INTERFACE I_DeserializerObjectForwardEnumerator EXTENDS I_Disposable

PROPERTY PUBLIC Current : I_Deserializer
GET
END_GET
END_PROPERTY

PROPERTY IsValid : BOOL
GET
END_GET
END_PROPERTY

PROPERTY Key : T_MAXSTRING
GET
END_GET
END_PROPERTY

METHOD MoveNext : BOOL
VAR_INPUT
END_VAR
END_METHOD

END_INTERFACE

(* stored: Version 1.1.0.1, ProductVersion 3.1.4024.12
   Itf I_DeserializerObjectForwardEnumerator: Id {4aa77d71-92a4-036e-397e-318ade50e4f8}
   Property Current: Id {c85a0a2e-7ad5-0667-211d-0f0eb5551b1d}
   Get Get: Id {dc71cbed-b22a-06bb-1cde-d3cef839c8cc}
   Property IsValid: Id {e0b342ed-ea59-00ab-0145-3d582b50d050}
   Get Get: Id {1adcd0c0-e8e5-03ae-0d04-9d5bad6bb5fd}
   Property Key: Id {166b0429-2001-0abb-3b8a-e0bee278bcc5}
   Get Get: Id {f06c18ae-1785-08a5-1551-518234def58e}
   Method MoveNext: Id {4574f2b1-7060-0cde-203a-71206c00cc4c} *)
